// TIA Portal project "rfid" (V16)

(* hardware
DEVICE "S7-1200 station_1"  S7-1200 Station
   slot 0: "Rack_0"  S7-1200 Rack  Rack  V1.0
   slot 1: "PLC_1"  CPU 1215C DC/DC/DC  6ES7 215-1AG40-0XB0  V4.4
DEVICE "PC station"  SIMATIC PC station
   slot 0: "PC station"  Rail  SIMATIC PC-Station  V1.0
      slot 125: "Stationmanager"  Station_Manager  V6.0.4
   slot 1: "IE general_1"  IE General  IE_CP  V8.2.0
   slot 2: "HMI_RT_1"  WinCC RT Advanced  6AV2 104-0xxxx-xxxx  16.0.0.0
      slot 33792: "Computer interface"  Host interface
*)

// ===== PLC "PLC_1"  CPU 1215C DC/DC/DC =====

VAR_GLOBAL   // PLC tag table "Default tag table"
   "Connect" AT %M15.0 : Bool;
   "send" AT %M15.1 : Bool;
   "Connection_established_trigger" AT %M15.2 : Bool;
   "Connection established" AT %M15.3 : Bool;
   "Connection_termination_trigger" AT %M15.4 : Bool;
   "Connection_terminated" AT %M15.5 : Bool;
   "Packet_sent_trig" AT %M16.0 : Bool;
   "Packed_sent" AT %M16.1 : Bool;
   "Clock_1Hz" AT %M0.5 : Bool;
   "System_Byte" AT %MB1 : Byte;
   "FirstScan" AT %M1.0 : Bool;
   "DiagStatusUpdate" AT %M1.1 : Bool;
   "AlwaysTRUE" AT %M1.2 : Bool;
   "AlwaysFALSE" AT %M1.3 : Bool;
   "Clock_Byte" AT %MB0 : Byte;
   "Clock_10Hz" AT %M0.0 : Bool;
   "Clock_5Hz" AT %M0.1 : Bool;
   "Clock_2.5Hz" AT %M0.2 : Bool;
   "Clock_2Hz" AT %M0.3 : Bool;
   "Clock_1.25Hz" AT %M0.4 : Bool;
   "Clock_0.625Hz" AT %M0.6 : Bool;
   "Clock_0.5Hz" AT %M0.7 : Bool;
   "Lifebit" AT %M100.0 : Bool;
   "received_trig" AT %M16.2 : Bool;
   "Tag_2" AT %M40.0 : Bool;
   "Tag_3" AT %M40.1 : Bool;
   "Tag_4" AT %M40.5 : Bool;
   "Tag_5" AT %M40.2 : Bool;
   "Tag_6" AT %M40.3 : Bool;
   "Tag_7" AT %M41.0 : Bool;
   "Tag_8" AT %M45.0 : Bool;
   "Clear mem" AT %M25.0 : Bool;
   "Tag_1" AT %M25.1 : Bool;
   "write_epc" AT %M15.6 : Bool;
END_VAR

DATA_BLOCK "Data_block_1"   // DB1
{ S7_Optimized_Access := 'TRUE' }
VERSION : 0.1
   VAR
      cmd_list : Array[0..6] of String;
      receive_arr : Array[0..250] of Char;
      received_epc : String;
      receive_arr_str : String;
      send_arr : Array[0..250] of Char;
      "set led" : Struct
         "0 1" : Array[0..1] of Char;
         "3" : Char := '_';
         "4" : Char := '0';
         "5" : Char := '0';
         "6" : Char := '_';
         "7" : Char := 'M';
         "8" : Char := 'N';
         "9" : Char := '_';
         "10 80" : Array[0..23] of String;
         "81 82" : Array[0..1] of Char;
      END_STRUCT;
      asd : UInt;
      strlen : UInt;
      frame_count : UInt;
      cmd_nr : UInt;
      ID1_rssi : String;
      ID2_rssi : String;
      ID1_val : String;
      ID2_val : String;
      empty_str : String;
      write_val : String;
   END_VAR
BEGIN
   "set led"."0 1"[0] := 'S';
   "set led"."0 1"[1] := 'L';
   "set led"."10 80"[0] := '00_';
   "set led"."10 80"[1] := '00_';
   "set led"."10 80"[2] := '00_';
   "set led"."10 80"[3] := '00_';
   "set led"."10 80"[4] := '00_';
   "set led"."10 80"[5] := '00_';
   "set led"."10 80"[6] := '01_';
   "set led"."10 80"[7] := '00_';
   "set led"."10 80"[8] := '00_';
   "set led"."10 80"[9] := '00_';
   "set led"."10 80"[10] := '00_';
   "set led"."10 80"[11] := '00_';
   "set led"."10 80"[12] := '00_';
   "set led"."10 80"[13] := '00_';
   "set led"."10 80"[14] := '00_';
   "set led"."10 80"[15] := '00_';
   "set led"."10 80"[16] := '00_';
   "set led"."10 80"[17] := '00_';
   "set led"."10 80"[18] := '00_';
   "set led"."10 80"[19] := '00_';
   "set led"."10 80"[20] := '00_';
   "set led"."10 80"[21] := '00_';
   "set led"."10 80"[22] := '00_';
   "set led"."10 80"[23] := '00';
   "set led"."81 82"[0] := '$R';
   "set led"."81 82"[1] := '$L';
   cmd_list[2] := 'SL_00_MN_01_01_01_01_01_01_01_01_01_01_01_01_01_01_01_01_01_01_01_01_01_01_01_01$R$L';
   cmd_list[0] := 'GM$R$L';
   cmd_list[1] := 'SL_00_AT_01_01_01_01_01_01_01_01_01_01_01_01_01_01_01_01_01_01_01_01_01_01_01_01$R$L';
   cmd_list[3] := 'SL_00_MN_00_00_00_00_00_00_00_00_00_00_00_00_00_00_00_00_00_00_00_00_00_00_00_00$R$L';
   cmd_list[4] := 'RP_01$R$L';
   cmd_list[5] := 'DI_01$R$L';
   cmd_list[6] := 'WP_01_2_11_2_AB$R$L';
END_DATA_BLOCK

// folder: System blocks/Program resources

DATA_BLOCK "IEC_Timer_0_DB"   // DB3
{ S7_Optimized_Access := 'TRUE' }
AUTHOR : Simatic
FAMILY : IEC
NAME : IEC_TMR
VERSION : 1.0
// stored: InstanceOfName IEC_TIMER
"IEC_TIMER"
BEGIN
END_DATA_BLOCK

DATA_BLOCK "PLC_1_Send_DB"   // DB4
{ S7_Optimized_Access := 'TRUE' }
AUTHOR : SIMATIC
FAMILY : MC7Plus
NAME : TC_IP_v4
VERSION : 1.0
// stored: InstanceOfName TCON_IP_v4
"TCON_IP_v4"
BEGIN
   ID := 1;
   InterfaceId := 64;
   RemotePort := 2000;
   ActiveEstablished := true;
   ConnectionType := 11;
   RemoteAddress.ADDR[1] := 192;
   RemoteAddress.ADDR[2] := 168;
   RemoteAddress.ADDR[4] := 79;
END_DATA_BLOCK

DATA_BLOCK "IEC_Timer_0_DB_1"   // DB8
{ S7_Optimized_Access := 'TRUE' }
AUTHOR : Simatic
FAMILY : IEC
NAME : IEC_TMR
VERSION : 1.0
// stored: InstanceOfName IEC_TIMER
"IEC_TIMER"
BEGIN
END_DATA_BLOCK

DATA_BLOCK "IEC_Counter_0_DB_1"   // DB9
{ S7_Optimized_Access := 'TRUE' }
AUTHOR : Simatic
FAMILY : IEC
NAME : UCNTR
VERSION : 1.2
// stored: InstanceOfName IEC_UCOUNTER
"IEC_UCOUNTER"
BEGIN
END_DATA_BLOCK

// folder: (top level)

FUNCTION "Block_2" : Void   // FC1, LAD
{ S7_Optimized_Access := 'TRUE' }
VERSION : 0.1
   VAR_TEMP   // added for the SCL form of the ladder/FBD networks
      _w1 : Bool;
      _w2 : Bool;
      _w3 : Bool;
      _w4 : Bool;
   END_VAR
BEGIN

REGION Network 1: tworzenie i usuwanie połączenia
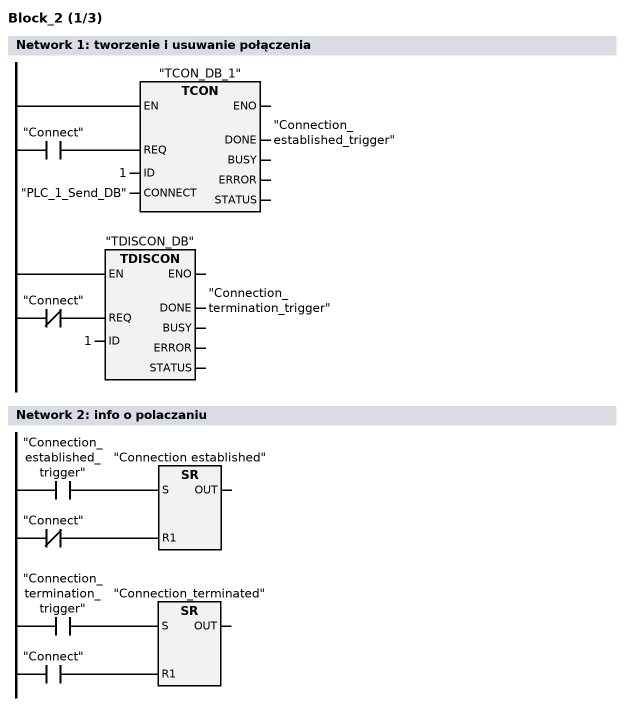
   "TCON_DB_1"(REQ := "Connect", ID := 1, CONNECT := "PLC_1_Send_DB", DONE => "Connection_established_trigger");   // TCON
   "TDISCON_DB"(REQ := NOT "Connect", ID := 1, DONE => "Connection_termination_trigger");   // TDISCON
END_REGION

REGION Network 2: info o polaczaniu
   RUNG wire#powerrail
      Contact( "Connection_established_trigger" )
      S_SR(operand := "Connection established", r1 := wire#w1)
   END_RUNG
   RUNG wire#powerrail
      I_Contact( "Connect" )
   END_RUNG wire#w1
   RUNG wire#powerrail
      Contact( "Connection_termination_trigger" )
      S_SR(operand := "Connection_terminated", r1 := wire#w2)
   END_RUNG
   RUNG wire#powerrail
      Contact( "Connect" )
   END_RUNG wire#w2
   // the same network as SCL:
   IF "Connection_established_trigger" THEN
       "Connection established" := TRUE;   // SR flip-flop
   END_IF;
   IF NOT "Connect" THEN "Connection established" := FALSE; END_IF;
   IF "Connection_termination_trigger" THEN
       "Connection_terminated" := TRUE;   // SR flip-flop
   END_IF;
   IF "Connect" THEN "Connection_terminated" := FALSE; END_IF;
END_REGION

REGION Network 3: wysylanie
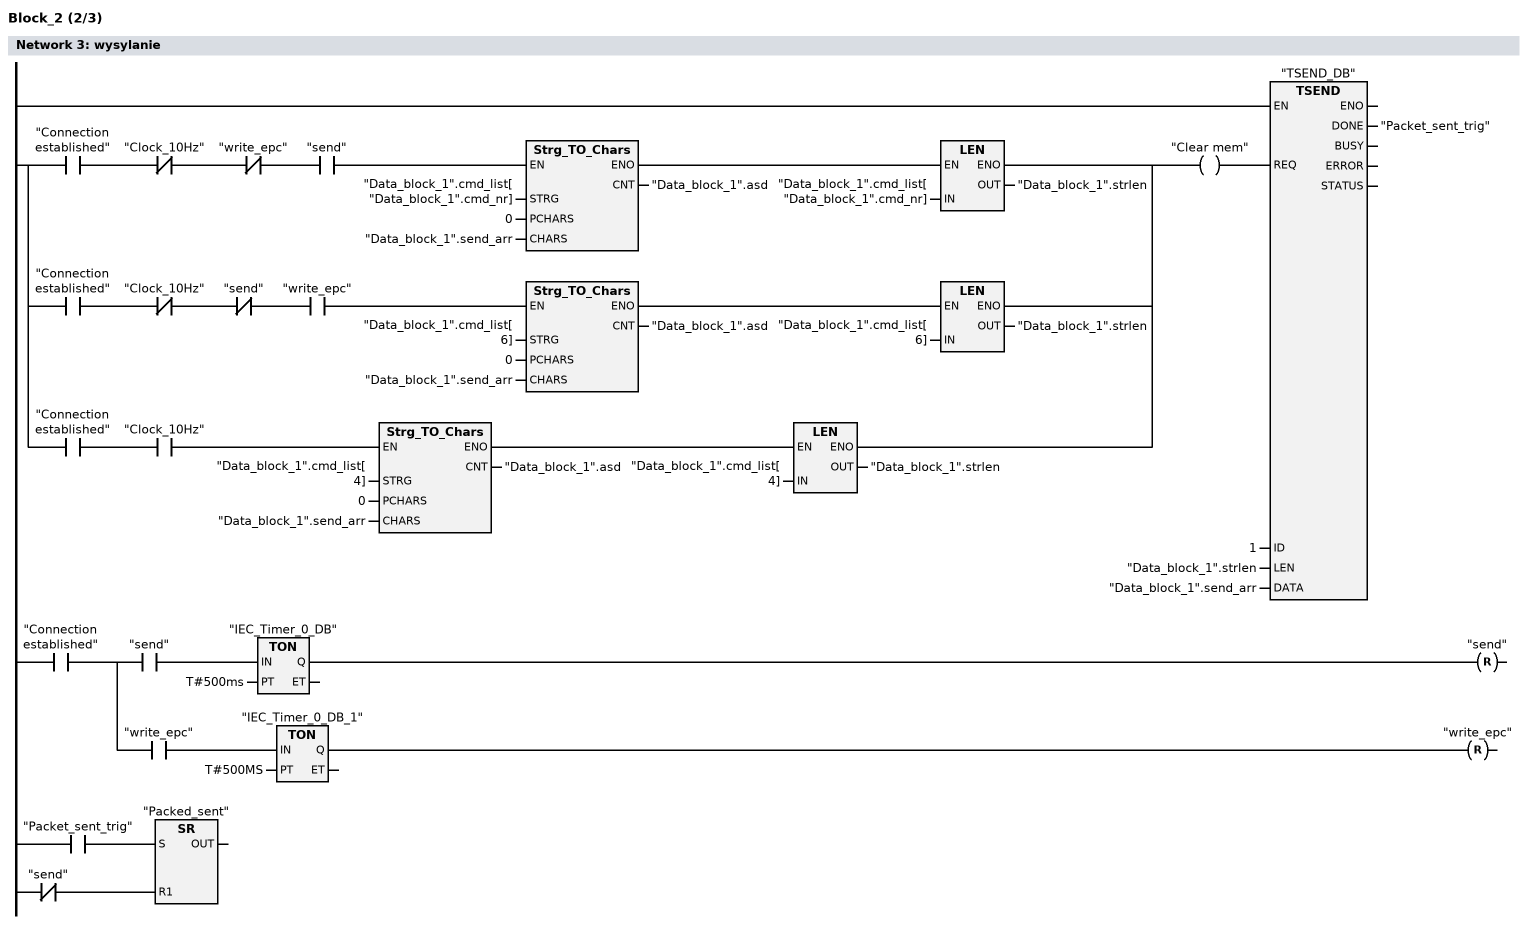
   // no SCL statement known for Strg_TO_Chars: written as a call
   // ENO of a box is taken as its EN; it also drops when the box reports an error
   #_w1 := "Connection established" AND NOT "Clock_10Hz" AND NOT "write_epc" AND "send";
   IF #_w1 THEN
       Strg_TO_Chars(Strg := "Data_block_1".cmd_list["Data_block_1".cmd_nr],
                     pChars := 0,
                     Chars := "Data_block_1".send_arr,
                     Cnt => "Data_block_1".asd);
       "Data_block_1".strlen := LEN(IN := "Data_block_1".cmd_list["Data_block_1".cmd_nr]);
   END_IF;
   #_w2 := "Connection established" AND NOT "Clock_10Hz" AND NOT "send" AND "write_epc";
   IF #_w2 THEN
       Strg_TO_Chars(Strg := "Data_block_1".cmd_list[6],
                     pChars := 0,
                     Chars := "Data_block_1".send_arr,
                     Cnt => "Data_block_1".asd);
       "Data_block_1".strlen := LEN(IN := "Data_block_1".cmd_list[6]);
   END_IF;
   #_w3 := "Connection established" AND "Clock_10Hz";
   IF #_w3 THEN
       Strg_TO_Chars(Strg := "Data_block_1".cmd_list[4],
                     pChars := 0,
                     Chars := "Data_block_1".send_arr,
                     Cnt => "Data_block_1".asd);
       "Data_block_1".strlen := LEN(IN := "Data_block_1".cmd_list[4]);
   END_IF;
   "Clear mem" := #_w1 OR #_w2 OR #_w3;
   "TSEND_DB"(REQ := "Clear mem",   // TSEND
              ID := 1,
              LEN := "Data_block_1".strlen,
              DATA := "Data_block_1".send_arr,
              DONE => "Packet_sent_trig");
   "IEC_Timer_0_DB".TON(IN := "Connection established" AND "send", PT := T#500ms);
   IF "IEC_Timer_0_DB".Q THEN "send" := FALSE; END_IF;
   "IEC_Timer_0_DB_1".TON(IN := "Connection established" AND "write_epc", PT := T#500MS);
   IF "IEC_Timer_0_DB_1".Q THEN "write_epc" := FALSE; END_IF;
   IF "Packet_sent_trig" THEN
       "Packed_sent" := TRUE;   // SR flip-flop
   END_IF;
   IF NOT "send" THEN "Packed_sent" := FALSE; END_IF;
END_REGION

REGION Network 4: odbieranie
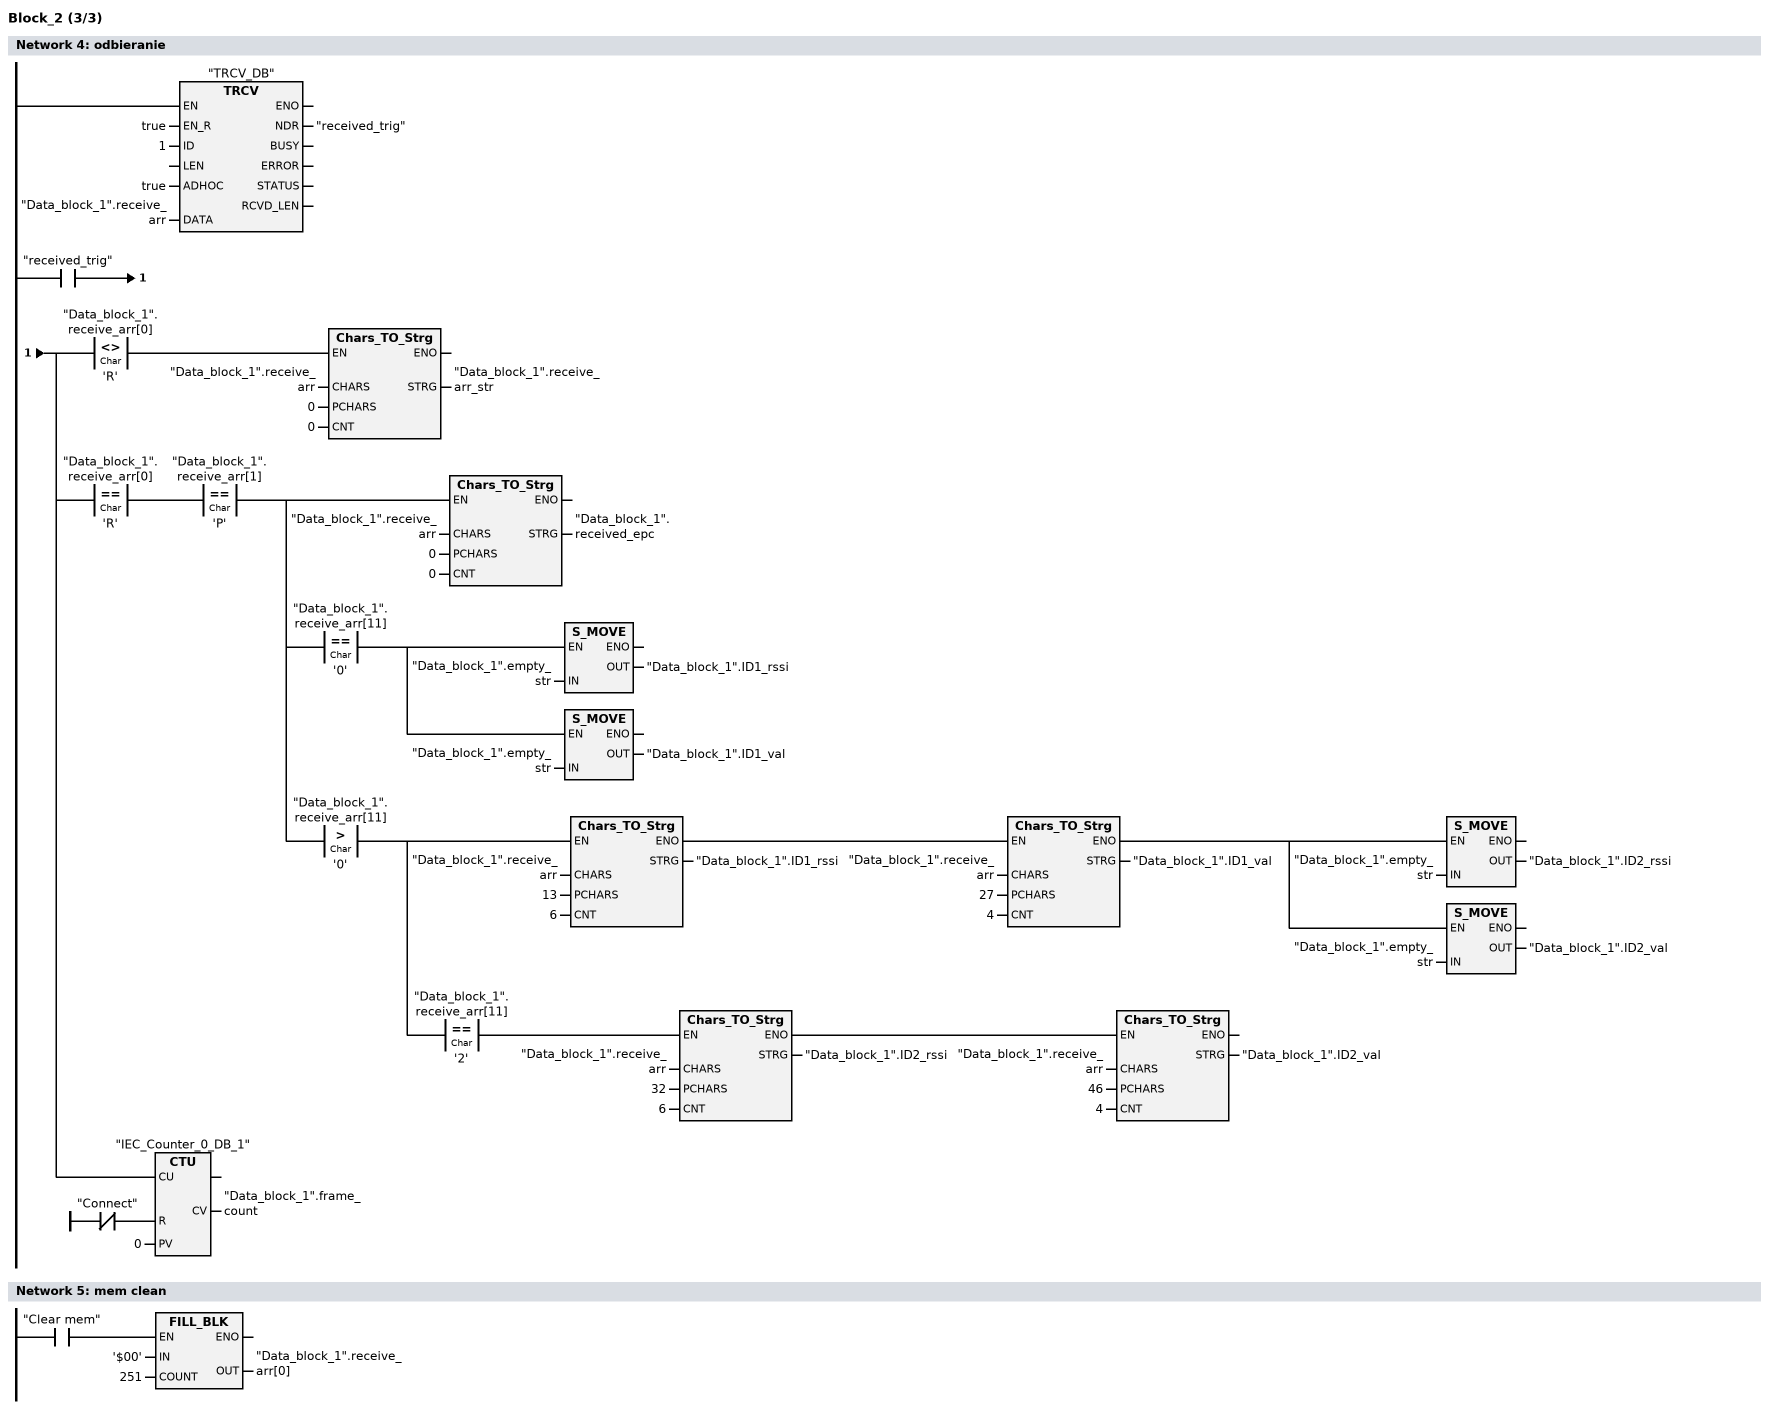
   // no SCL statement known for Chars_TO_Strg: written as a call
   // ENO of a box is taken as its EN; it also drops when the box reports an error
   "TRCV_DB"(EN_R := true, ID := 1, ADHOC := true, DATA := "Data_block_1".receive_arr, NDR => "received_trig");   // TRCV
   #_w1 := "received_trig";
   IF "received_trig" AND ("Data_block_1".receive_arr[0] <> 'R') THEN
       Chars_TO_Strg(Chars := "Data_block_1".receive_arr,
                     pChars := 0,
                     Cnt := 0,
                     Strg => "Data_block_1".receive_arr_str);
   END_IF;
   #_w2 := #_w1 AND ("Data_block_1".receive_arr[0] = 'R') AND ("Data_block_1".receive_arr[1] = 'P');
   IF #_w2 THEN
       Chars_TO_Strg(Chars := "Data_block_1".receive_arr,
                     pChars := 0,
                     Cnt := 0,
                     Strg => "Data_block_1".received_epc);
   END_IF;
   IF #_w2 AND ("Data_block_1".receive_arr[11] = '0') THEN
       "Data_block_1".ID1_rssi := "Data_block_1".empty_str;
       "Data_block_1".ID1_val := "Data_block_1".empty_str;
   END_IF;
   #_w3 := #_w2 AND ("Data_block_1".receive_arr[11] > '0');
   IF #_w3 THEN
       Chars_TO_Strg(Chars := "Data_block_1".receive_arr, pChars := 13, Cnt := 6, Strg => "Data_block_1".ID1_rssi);
       Chars_TO_Strg(Chars := "Data_block_1".receive_arr, pChars := 27, Cnt := 4, Strg => "Data_block_1".ID1_val);
       "Data_block_1".ID2_rssi := "Data_block_1".empty_str;
       "Data_block_1".ID2_val := "Data_block_1".empty_str;
   END_IF;
   #_w4 := #_w3 AND ("Data_block_1".receive_arr[11] = '2');
   IF #_w4 THEN
       Chars_TO_Strg(Chars := "Data_block_1".receive_arr, pChars := 32, Cnt := 6, Strg => "Data_block_1".ID2_rssi);
       Chars_TO_Strg(Chars := "Data_block_1".receive_arr, pChars := 46, Cnt := 4, Strg => "Data_block_1".ID2_val);
   END_IF;
   "IEC_Counter_0_DB_1".CTU(CU := #_w1, R := NOT "Connect", PV := 0, CV => "Data_block_1".frame_count);
END_REGION

REGION Network 5: mem clean
   RUNG wire#powerrail
      Contact( "Clear mem" )
      FillBlockI(in := '$00', count := 251, out => "Data_block_1".receive_arr[0])
   END_RUNG
   // the same network as SCL:
   IF "Clear mem" THEN FILL_BLK(IN := '$00', COUNT := 251, OUT => "Data_block_1".receive_arr[0]); END_IF;
END_REGION
END_FUNCTION

ORGANIZATION_BLOCK "Main"   // OB1, LAD, ProgramCycle
TITLE = "Main Program Sweep (Cycle)"
{ S7_Optimized_Access := 'TRUE' }
VERSION : 0.1
   VAR_INPUT
      Initial_Call : Bool;   // Initial call of this OB
      Remanence : Bool;   // =True, if remanent data are available
   END_VAR
BEGIN

REGION Network 1
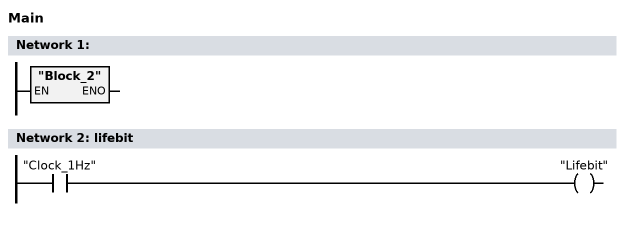
   RUNG wire#powerrail
      "Block_2"()
   END_RUNG
   // the same network as SCL:
   "Block_2"();
END_REGION

REGION Network 2: lifebit
   RUNG wire#powerrail
      Contact( "Clock_1Hz" )
      Coil( "Lifebit" )
   END_RUNG
   // the same network as SCL:
   "Lifebit" := "Clock_1Hz";
END_REGION
END_ORGANIZATION_BLOCK

(* ===== HMI "HMI_RT_1" =====
system functions are stored by id; their names below are inferred from use
connection "HMI_Connection_1": ETHERNET, S7_1200_OMS

HMI tags "Default tag table"
   "Lifebit" : Bool = PLC Lifebit AT %M100.0, 100 ms
   "Connect" : Bool = PLC Connect AT %M15.0, 100 ms
   "Connection establisheda" : Bool = PLC "Connection established" AT %M15.3, 500 ms
   "send1" : Bool = PLC send AT %M15.1, 100 ms
   "Packed_sent1" : Bool = PLC Packed_sent AT %M16.1, 100 ms
   "receive_str" : String[254] = PLC Data_block_1.receive_arr_str AT %DB1.DBX0.0, 100 ms
   "Data_block_1_frame_count" : UInt = PLC Data_block_1.frame_count, 100 ms
   "Data_block_1_testint" : UInt = PLC Data_block_1.cmd_nr, 100 ms
   "Data_block_1_received_epc" : String[254] = PLC Data_block_1.received_epc, 100 ms
   "Data_block_1_ID1_rssi" : String[254] = PLC Data_block_1.ID1_rssi, 100 ms
   "Data_block_1_ID2_rssi" : String[254] = PLC Data_block_1.ID2_rssi, 100 ms
   "Data_block_1_ID1_val" : String[254] = PLC Data_block_1.ID1_val, 100 ms
   "Data_block_1_ID2_val" : String[254] = PLC Data_block_1.ID2_val, 100 ms
   "write_epc" : Bool = PLC write_epc AT %M15.6, 100 ms
   "Data_block_1_write_val" : String[254] = PLC Data_block_1.write_val, 100 ms

text list "Text_list_1": 0 'Get mac'; 2 'Set all led on'; 3 'Set all led off'; 1 'Led mode auto'; 5 'Diagnostic info'

screen "Screen_1" 1024x768
   Circle "Circle_1" at 1,1 size 44x44
      Appearance <- "Lifebit"
   Button "Button_1" at 10,96 size 96x32; TextOff 'Connect'
      on Click: InvertBit("Connect")
   Circle "Circle_2" at 113,96 size 32x32
      Appearance <- "Connection establisheda"
   Button "Button_2" at 10,145 size 154x32; TextOff 'Send cmd'
      on Click: SetBit("send1")
   Circle "Circle_3" at 175,145 size 32x32
      Appearance <- "Packed_sent1"
   IOField "I/O field_1" at 450,104 size 571x35; FormatPattern ??????????????????????????????????????????????????????????????????????????????????????????????????????????????????????????????????????????????????????????????????????????????????????????????????????????????????????????????????????????????????????????????
      ProcessValue <- "receive_str"
   Group "Group" at 314,96 size 130x48
   Group "Group_1" at 315,156 size 129x48
   IOField "I/O field_2" at 452,162 size 76x35; FormatPattern 99999
      ProcessValue <- "Data_block_1_frame_count"
   SymbolicIOField "Symbolic I/O field_1" at 9,182 size 202x32; TextOff '0'; TextOn '1'; TextList "Text_list_1"
      ProcessValue <- "Data_block_1_testint"
   IOField "I/O field_3" at 150,313 size 873x35; FormatPattern ??????????????????????????????????????????????????????????????????????????????????????????????????????????????????????????????????????????????????????????????????????????????????????????????????????????????????????????????????????????????????????????????
      ProcessValue <- "Data_block_1_received_epc"
   Group "Group_2" at 0,305 size 149x48
   Group "Group_3" at 171,383 size 143x48
   Group "Group_4" at 380,383 size 147x48
   IOField "I/O field_4" at 204,452 size 96x32; FormatPattern ??????
      ProcessValue <- "Data_block_1_ID1_rssi"
   IOField "I/O field_5" at 408,452 size 96x32; FormatPattern ??????
      ProcessValue <- "Data_block_1_ID2_rssi"
   Group "Group_5" at 60,450 size 77x31
   IOField "I/O field_6" at 204,501 size 96x32; FormatPattern ??????????????????????????????
      ProcessValue <- "Data_block_1_ID1_val"
   IOField "I/O field_7" at 408,501 size 96x32; FormatPattern ??????????????????????????????
      ProcessValue <- "Data_block_1_ID2_val"
   Group "Group_6" at 61,497 size 76x33
   Button "Button_3" at 211,589 size 96x32; TextOff 'Write'
      on Click: SetBit("write_epc")
   IOField "I/O field_8" at 387,589 size 96x32; FormatPattern ????
      ProcessValue <- "Data_block_1_write_val"
   IOField "I/O field_9" at 211,631 size 96x32; FormatPattern ????
      ProcessValue <- "Data_block_1_write_val"
   TextField "Text field_8" at 414,567 size 74x22; Text 'INPUT'
   TextField "Text field_1" at 336,110 size 94x22; Text 'Received'
   TextField "Text field_2" at 337,170 size 96x22; Text 'Frame nr'
   TextField "Text field_3" at 10,319 size 139x22; Text 'Received EPC'
   TextField "Text field_4" at 227,397 size 65x22; Text 'ID1'
   TextField "Text field_5" at 437,397 size 85x22; Text 'ID2'
   TextField "Text field_6" at 68,457 size 63x22; Text 'RSSI'
   TextField "Text field_7" at 68,505 size 66x22; Text 'value'
*)